{attribute 'GeneratedUsingTerminal: EL6001-0000-0020'}
{attribute addProperty BoxType "EL6001-0000-0020"}
{attribute addProperty Id "StatusAT %I*USINT1Data_InAT %I*ARRAY[0..4] OF USINT5"}
{attribute addProperty CRC "3276876527"}
{attribute addProperty Size "6"}
TYPE Inputs_37C8E74C :
STRUCT
	{attribute addProperty Name "Status"}
	Status AT %I* : USINT;
	{attribute addProperty Name "Data_In"}
	Data_In AT %I* : ARRAY[0..4] OF USINT;
END_STRUCT
END_TYPE

(* stored: Version 1.2.0.0, ProductVersion 3.1.4024.9
   DUT Inputs_37C8E74C: Id {949f1f79-3462-461d-8cda-c1f2a40c36b1} *)
